// Interface that defines the arithmetic operations for a time instance.
INTERFACE I_TimeInstanceArithmetics EXTENDS __SYSTEM.IQueryInterface

END_INTERFACE

(* stored: Version 1.1.0.1
   Itf I_TimeInstanceArithmetics: Id {e0643f71-d721-0ade-15fb-ada06a838498} *)
